{attribute addProperty BoxType "EJ7211-0010-0026"}
{attribute addProperty Id "PositionAT %I*UDINT324"}
{attribute addProperty CRC "3129649648"}
{attribute addProperty SizeInBites "32"}
{attribute addProperty SizeInBytes "4"}
TYPE FB_Position_BA8AA9F0 :
STRUCT
	{attribute addProperty Name "Position"}
	Position AT %I* : UDINT;
END_STRUCT
END_TYPE

(* stored: Version 1.2.0.0, ProductVersion 3.1.4024.9
   DUT FB_Position_BA8AA9F0: Id {c6b00e24-5139-47c7-a9b0-11536032eea9} *)
